PROGRAM MAIN
VAR
	testInt32ToROS AT %Q* :DINT :=0 ;
	testBoolToROS AT %Q*:BOOL :=TRUE;
	testInt32FromROS AT %I* :DINT :=0;
	testBoolFromROS AT %I*:BOOL:=FALSE;
END_VAR

testInt32ToROS := testInt32ToROS+1;

END_PROGRAM

(* stored: Version 1.1.0.1
   POU MAIN: Id {29449686-51f8-4ee2-a45f-7ec2ea18fd3d}, SpecialFunc None *)
